FUNCTION_BLOCK Q_ObjEnableDisable_AB (* Command enable/disable object with AB adapter (BYTE) *)
  (* Standard: 61499-2; Description: Copyright (c) 2026 Meisterschulen am Ostbahnhof This program and the accompanying materials are made available under the terms of the Eclipse Public License 2.0 which is available at https://www.eclipse.org/legal/epl-2.0/ SPDX-License-Identifier: EPL-2.0 *)
  (* Version 1.0, 2026-04-24, Franz Höpfinger, Meisterschulen am Ostbahnhof, AB adapter wrapper for Q_ObjEnableDisable *)
  PACKAGE isobus::UT::Q;
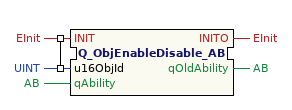
  EVENT_INPUT
    INIT : EInit WITH u16ObjId; (* Service Initialization *)
  END_EVENT
  EVENT_OUTPUT
    INITO : EInit; (* Initialization Confirm *)
  END_EVENT
  VAR_INPUT
    u16ObjId : UINT; (* Object ID *)
  END_VAR
  SOCKETS
    qAbility : adapter::types::unidirectional::AB; (* 0 == disable, 1 == enable, 0xFF == undefined *)
  END_SOCKETS
  PLUGS
    qOldAbility : adapter::types::unidirectional::AB; (* 0 == disable, 1 == enable, 0xFF == undefined *)
  END_PLUGS
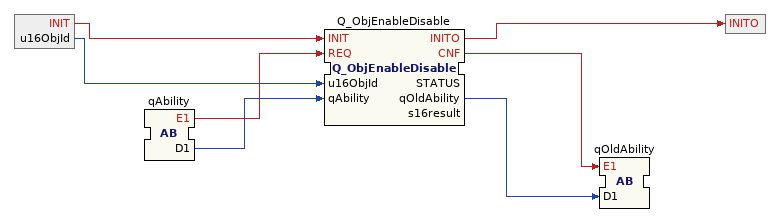
  FBS
    Q_ObjEnableDisable : isobus::UT::Q::Q_ObjEnableDisable;
  END_FBS
  EVENT_CONNECTIONS
    INIT TO Q_ObjEnableDisable.INIT;
    Q_ObjEnableDisable.INITO TO INITO;
    qAbility.E1 TO Q_ObjEnableDisable.REQ;
    Q_ObjEnableDisable.CNF TO qOldAbility.E1;
  END_CONNECTIONS
  DATA_CONNECTIONS
    u16ObjId TO Q_ObjEnableDisable.u16ObjId;
    qAbility.D1 TO Q_ObjEnableDisable.qAbility;
    Q_ObjEnableDisable.qOldAbility TO qOldAbility.D1;
  END_CONNECTIONS
END_FUNCTION_BLOCK
